(* PLC project Sin nombre, Desconocido Sin nombre 1 *)
(* stored: creationDateTime 2024-11-18T12:32:42, modificationDateTime 2024-11-20T12:05:53 *)

PROGRAM light_control
  VAR
    stairs_light AT %QX0.0 : BOOL;  (* Light switch turns on with true value *)
    lights_buttons_state AT %IX0.0 : BOOL;  (* Variable that indicates the state of lights according the buttons actions *)
    stairs_pir_sensor AT %IX0.1 : BOOL;  (* Passive Infrared Sensor detects persons arriving the stairs *)
    control_button_down AT %IX0.2 : BOOL;  (* Press button located down the stairs *)
    control_button_up AT %IX0.3 : BOOL;  (* Press button located up the stairs *)
  END_VAR
  VAR
    TOF0 : TOF;  (* Temporizador que marca el tiempo de encendido de la luz *)
  END_VAR
  VAR  (* added by the conversion: wires and edge detectors of the diagram *)
    R_TRIG1 : R_TRIG;
    R_TRIG2 : R_TRIG;
    R_TRIG3 : R_TRIG;
  END_VAR

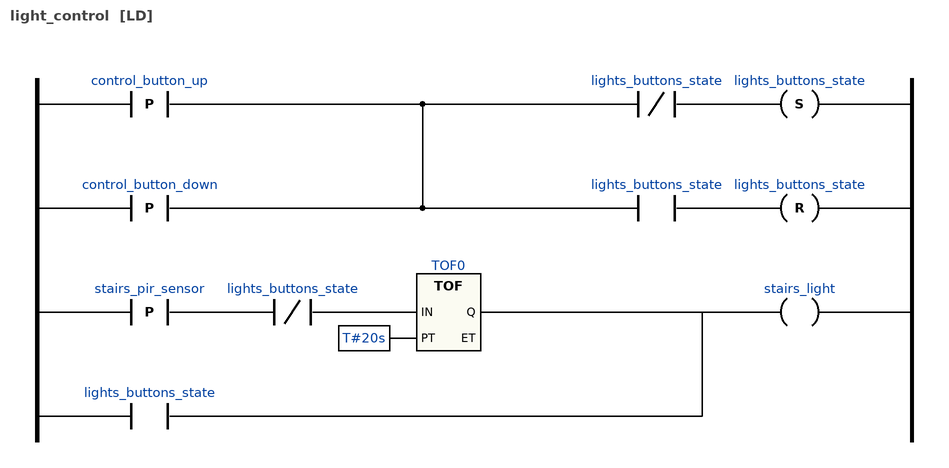
(* LD diagram, written out as Structured Text *)
R_TRIG1(CLK := control_button_down);
R_TRIG2(CLK := control_button_up);
IF (R_TRIG1.Q OR R_TRIG2.Q) AND NOT lights_buttons_state THEN lights_buttons_state := TRUE; END_IF;
IF (R_TRIG2.Q OR R_TRIG1.Q) AND lights_buttons_state THEN lights_buttons_state := FALSE; END_IF;
R_TRIG3(CLK := stairs_pir_sensor);
TOF0(IN := R_TRIG3.Q AND NOT lights_buttons_state, PT := T#20s);
stairs_light := TOF0.Q OR lights_buttons_state;
END_PROGRAM

CONFIGURATION Config0
  RESOURCE Res0 ON PLC
    TASK task0(INTERVAL := T#20ms, PRIORITY := 0);
    PROGRAM instance0 WITH task0 : light_control;
  END_RESOURCE
END_CONFIGURATION
